PROGRAM _02_Config_TEMP
VAR
	
	wTiempoPurga: WORD;
	ExisteValvPurga: BOOL;
END_VAR

(*-------------------------------------------------------------------------------------------------------*)

//Cargar valor pt-100
Mc._02_TEMP.rMacTemperature := Mc._02_TEMP.s065_Reg.rValue;

mc._02_TEMP.s065_Reg();

(* Activa Fallo PT100*)
Mc._02_TEMP.xPT100Failure := (Mc._02_TEMP.rMacTemperature >= 150) OR (Mc._02_TEMP.rMacTemperature <= 0);
///---------------------------------------------------------------------------------------------------------------

//Maxima diferencia 5 ºC
(*
Mc._02_TEMP.xMaxDifTemp := (F_TERMOREG.  AND ( Mc._02_TEMP.rMacTemperature > (Mc._02_TEMP.rTempImp+5) ) ) OR
						(F_TERMOREG.Termo.AiguaRefredament  AND ( Mc._02_TEMP.rMacTemperature < (Mc._02_TEMP.rTempImp-5) ) )	;

*)

END_PROGRAM

(* stored: Version 1.1.0.1, ProductVersion 3.1.4024.10
   POU _02_Config_TEMP: Id {efc90374-b168-4e5c-9a8a-07fc47a45383}, SpecialFunc None *)
